KUKA KRL data list: dai_math_library.dat

&ACCESS RVO6
&REL 18
&COMMENT daimler_mathematic_library
&USER PKL_AST
&PARAM version = 2.0
DEFDAT DAI_MATH_LIBRARY PUBLIC

;FOLD nearPos

;Toleranzwerte für nearE6Pos
DECL E6POS MaxPosTol={X 2.0,Y 2.0,Z 2.0,A 1.0,B 1.0,C 1.0,S 0,T 0,E1 2.0,E2 2.0,E3 2.0,E4 2.0,E5 2.0,E6 2.0}
;Toleranzwerte für nearE6Axis
DECL E6AXIS MaxAxisTol={A1 1.0,A2 1.0,A3 1.0,A4 1.0,A5 1.0,A6 1.0,E1 2.0,E2 2.0,E3 2.0,E4 2.0,E5 2.0,E6 2.0}

;ENDFOLD



ENDDAT
